# EPICS autosave request: autosave/galil_dmc_ctrl.req
$(P)LIMITTYPE_CMD
$(P)HOMETYPE_CMD
$(P)ECATNETWORK_CMD
$(P)DEFER_CMD
$(P)UPLOAD_CMD
$(P)DEFER_MODE_CMD
$(P)COORDSYS_CMD
$(P)OC1START_CMD
$(P)OC1INCR_CMD
$(P)OC1AXIS_CMD
$(P)OC2START_CMD
$(P)OC2INCR_CMD
$(P)OC2AXIS_CMD
$(P)SEND_STR_CMD
